FUNCTION_BLOCK FB_SchmittTriggerConsumer
VAR
    trigger : T1SchmittTrigger_Plc.FB_SchmittTrigger;
    bLastState : BOOL;
END_VAR

trigger(fInput := 0.5);
bLastState := trigger.Step();

END_FUNCTION_BLOCK

(* stored: Version 1.1.0.1
   POU FB_SchmittTriggerConsumer: Id {890d6316-6981-48a6-bd44-01e20a89a47a}, SpecialFunc None *)
